FUNCTION_BLOCK E_MERGE2
  (* Version 1.0, 2005-05-11, Goran Cengic, Chalmers *)
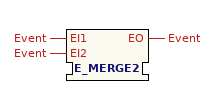
  EVENT_INPUT
    EI1;
    EI2;
  END_EVENT
  EVENT_OUTPUT
    EO;
  END_EVENT
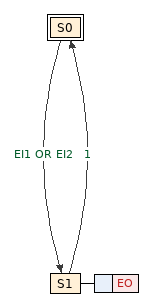
  EC_STATES
    S0;
    S1 : -> EO;
  END_STATES
  EC_TRANSITIONS
    S0 TO S1 := EI1 OR EI2;
    S1 TO S0 := 1;
  END_TRANSITIONS
END_FUNCTION_BLOCK
